// SIMATIC S7-200 SMART project (STEP 7-Micro/WIN SMART), CPU CR30s

ORGANIZATION_BLOCK MAIN:OB1
TITLE=Program Comments
BEGIN
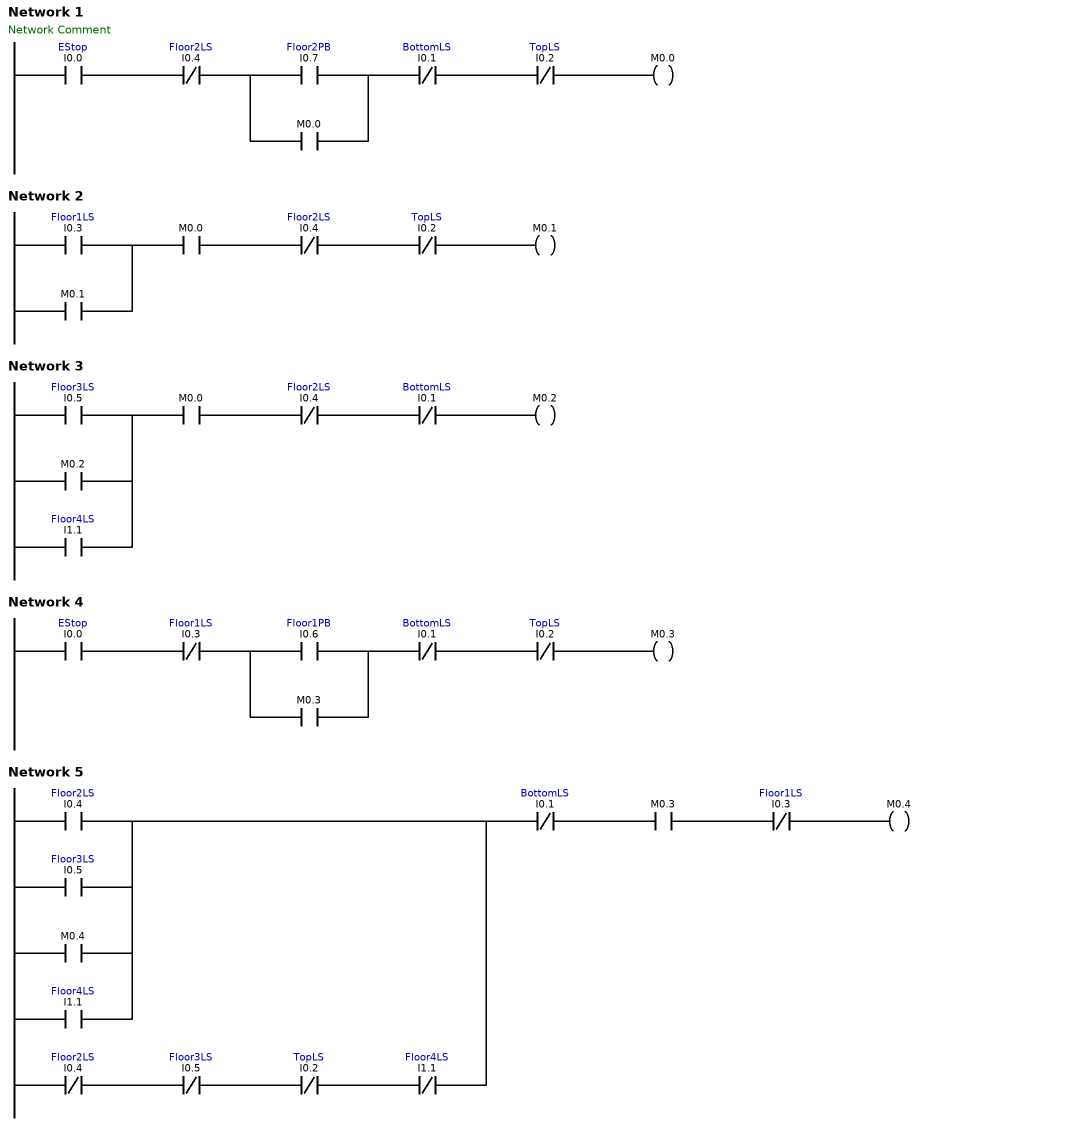
Network 1
// Network Comment
LD     EStop:I0.0
AN     Floor2LS:I0.4
LD     Floor2PB:I0.7
O      M0.0
ALD
AN     BottomLS:I0.1
AN     TopLS:I0.2
=      M0.0
Network 2
LD     Floor1LS:I0.3
O      M0.1
A      M0.0
AN     Floor2LS:I0.4
AN     TopLS:I0.2
=      M0.1
Network 3
LD     Floor3LS:I0.5
O      M0.2
O      Floor4LS:I1.1
A      M0.0
AN     Floor2LS:I0.4
AN     BottomLS:I0.1
=      M0.2
Network 4
LD     EStop:I0.0
AN     Floor1LS:I0.3
LD     Floor1PB:I0.6
O      M0.3
ALD
AN     BottomLS:I0.1
AN     TopLS:I0.2
=      M0.3
Network 5
LD     Floor2LS:I0.4
O      Floor3LS:I0.5
O      M0.4
O      Floor4LS:I1.1
LDN    Floor2LS:I0.4
AN     Floor3LS:I0.5
AN     TopLS:I0.2
AN     Floor4LS:I1.1
OLD
AN     BottomLS:I0.1
A      M0.3
AN     Floor1LS:I0.3
=      M0.4
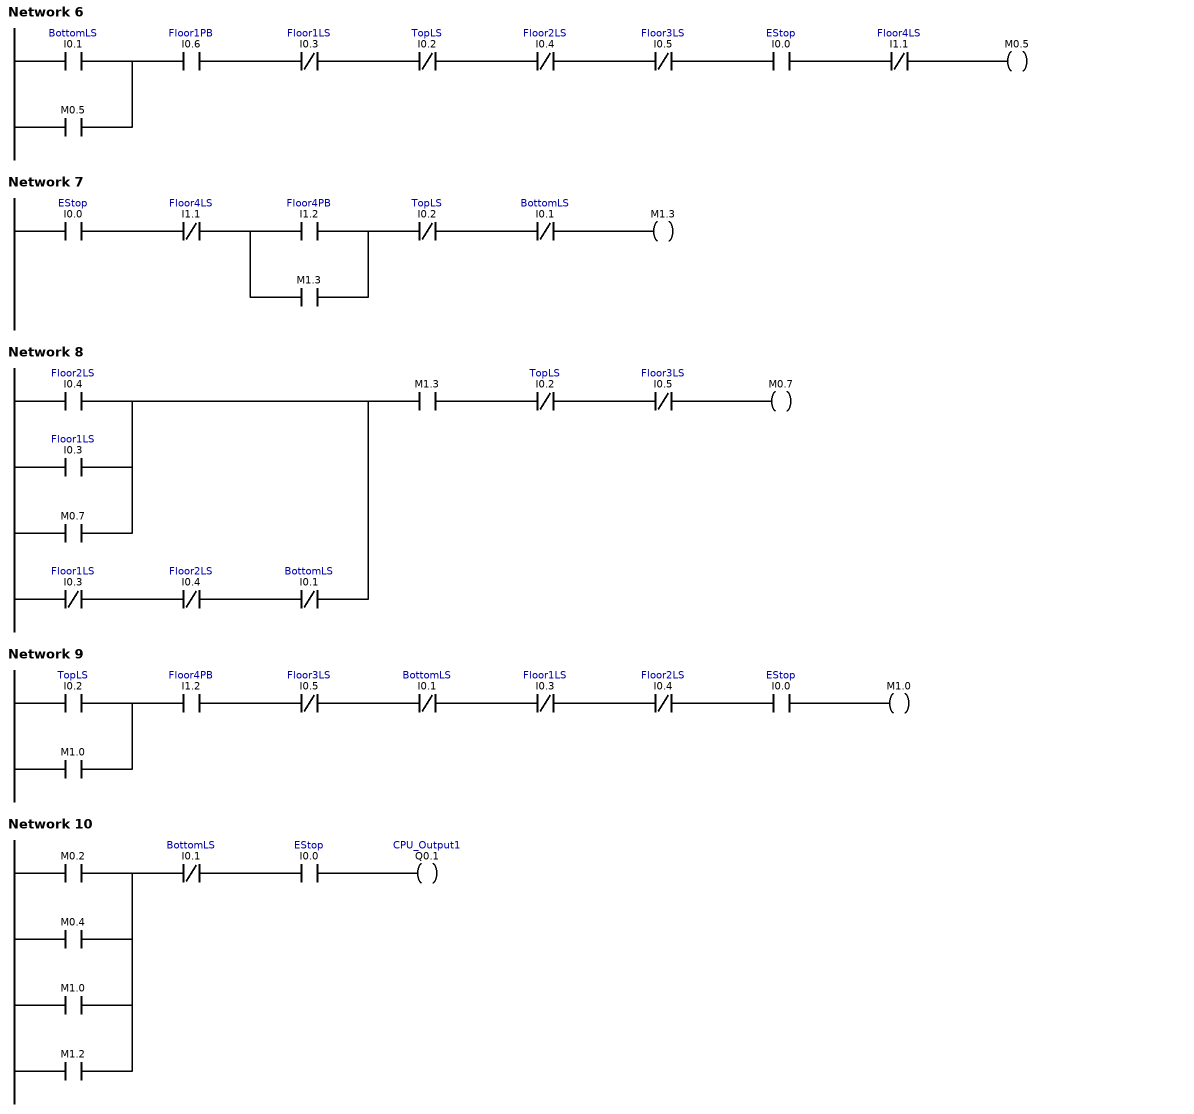
Network 6
LD     BottomLS:I0.1
O      M0.5
A      Floor1PB:I0.6
AN     Floor1LS:I0.3
AN     TopLS:I0.2
AN     Floor2LS:I0.4
AN     Floor3LS:I0.5
A      EStop:I0.0
AN     Floor4LS:I1.1
=      M0.5
Network 7
LD     EStop:I0.0
AN     Floor4LS:I1.1
LD     Floor4PB:I1.2
O      M1.3
ALD
AN     TopLS:I0.2
AN     BottomLS:I0.1
=      M1.3
Network 8
LD     Floor2LS:I0.4
O      Floor1LS:I0.3
O      M0.7
LDN    Floor1LS:I0.3
AN     Floor2LS:I0.4
AN     BottomLS:I0.1
OLD
A      M1.3
AN     TopLS:I0.2
AN     Floor3LS:I0.5
=      M0.7
Network 9
LD     TopLS:I0.2
O      M1.0
A      Floor4PB:I1.2
AN     Floor3LS:I0.5
AN     BottomLS:I0.1
AN     Floor1LS:I0.3
AN     Floor2LS:I0.4
A      EStop:I0.0
=      M1.0
Network 10
LD     M0.2
O      M0.4
O      M1.0
O      M1.2
AN     BottomLS:I0.1
A      EStop:I0.0
=      CPU_Output1:Q0.1
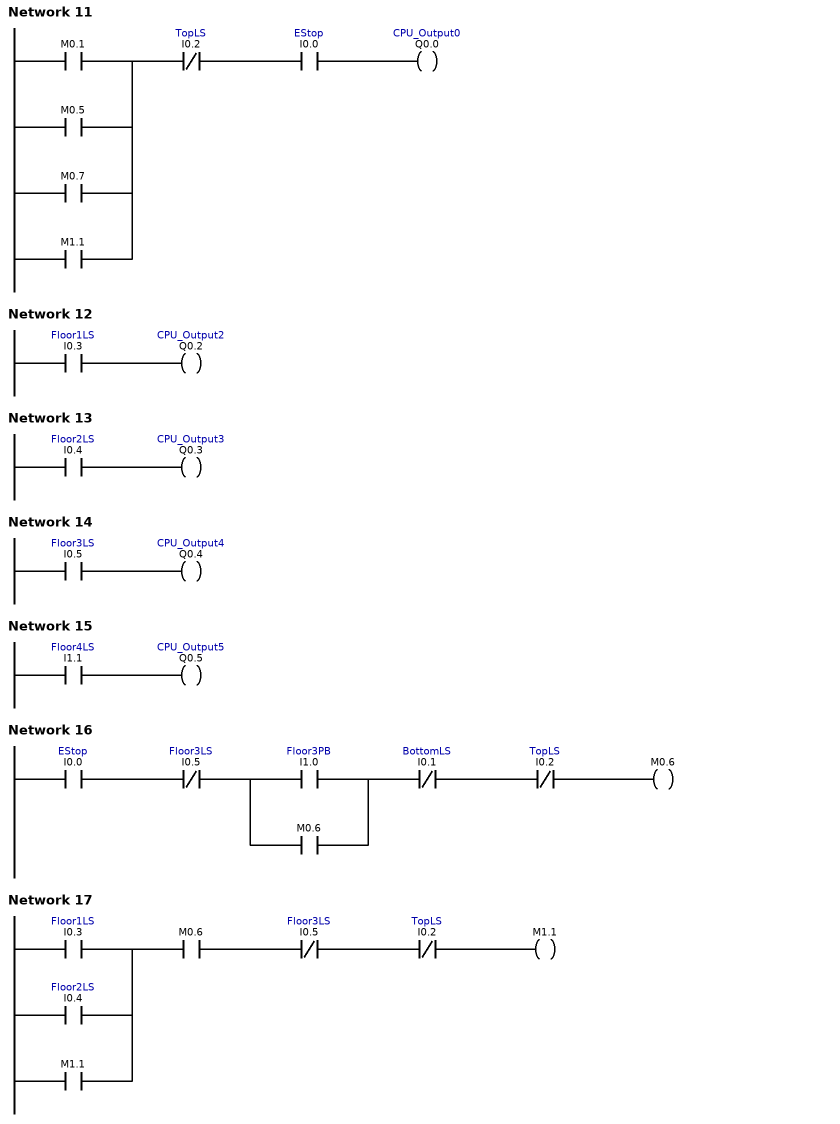
Network 11
LD     M0.1
O      M0.5
O      M0.7
O      M1.1
AN     TopLS:I0.2
A      EStop:I0.0
=      CPU_Output0:Q0.0
Network 12
LD     Floor1LS:I0.3
=      CPU_Output2:Q0.2
Network 13
LD     Floor2LS:I0.4
=      CPU_Output3:Q0.3
Network 14
LD     Floor3LS:I0.5
=      CPU_Output4:Q0.4
Network 15
LD     Floor4LS:I1.1
=      CPU_Output5:Q0.5
Network 16
LD     EStop:I0.0
AN     Floor3LS:I0.5
LD     Floor3PB:I1.0
O      M0.6
ALD
AN     BottomLS:I0.1
AN     TopLS:I0.2
=      M0.6
Network 17
LD     Floor1LS:I0.3
O      Floor2LS:I0.4
O      M1.1
A      M0.6
AN     Floor3LS:I0.5
AN     TopLS:I0.2
=      M1.1
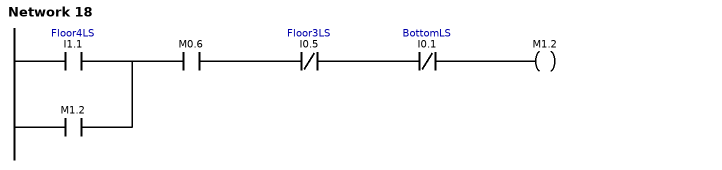
Network 18
LD     Floor4LS:I1.1
O      M1.2
A      M0.6
AN     Floor3LS:I0.5
AN     BottomLS:I0.1
=      M1.2
END_ORGANIZATION_BLOCK
